// TIA Portal V19 export
FUNCTION_BLOCK "TYPIC_C103_IF_HVI"   // FB20, FBD
TITLE = TYPIC_C103_IF_HVI: ALSB
{ S7_Optimized_Access := 'TRUE' }
AUTHOR : OCOTECH
FAMILY : Typical
NAME : C103.701
// Logisch Object Besturing: C103.802
// 
// De interne functie laagspanningsverdeelbord verzorgt de bewaking van een laagspanningsverdeelbord.
// stored: MemoryReserve 10, SetENOAutomatically false
   VAR_INPUT
      EXT_AUT { ExternalAccessible := 'False'; ExternalVisible := 'False'; ExternalWritable := 'False'} : Bool;   // Externe (hoofd) beveiliging (1 = OK)
      EXT_HW { ExternalAccessible := 'False'; ExternalVisible := 'False'; ExternalWritable := 'False'} : Bool;   // Sturings hardware (PLC) bewaking (1 = OK)
      IN_PWR1 { ExternalAccessible := 'False'; ExternalVisible := 'False'; ExternalWritable := 'False'} : Real;   // Actief vermogen
      IN_PWR2 { ExternalAccessible := 'False'; ExternalVisible := 'False'; ExternalWritable := 'False'} : Real;   // Reactief vermogen
      IN_SPA_1 { ExternalAccessible := 'False'; ExternalVisible := 'False'; ExternalWritable := 'False'} : Real;   // Spanningsniveau lijn 1
      IN_SPA_2 { ExternalAccessible := 'False'; ExternalVisible := 'False'; ExternalWritable := 'False'} : Real;   // Spanningsniveau lijn 2
      IN_SPA_3 { ExternalAccessible := 'False'; ExternalVisible := 'False'; ExternalWritable := 'False'} : Real;   // Spanningsniveau lijn 3
      IN_SPA_4 { ExternalAccessible := 'False'; ExternalVisible := 'False'; ExternalWritable := 'False'} : Real;   // Lijnspanning L1-L2
      IN_SPA_5 { ExternalAccessible := 'False'; ExternalVisible := 'False'; ExternalWritable := 'False'} : Real;   // Lijnspanning L2-L3
      IN_SPA_6 { ExternalAccessible := 'False'; ExternalVisible := 'False'; ExternalWritable := 'False'} : Real;   // Lijnspanning L1-L3
      IN_STR_1 { ExternalAccessible := 'False'; ExternalVisible := 'False'; ExternalWritable := 'False'} : Real;   // Stroom lijn 1
      IN_STR_2 { ExternalAccessible := 'False'; ExternalVisible := 'False'; ExternalWritable := 'False'} : Real;   // Stroom lijn 2
      IN_STR_3 { ExternalAccessible := 'False'; ExternalVisible := 'False'; ExternalWritable := 'False'} : Real;   // Stroom lijn 3
      IN_STR_4 { ExternalAccessible := 'False'; ExternalVisible := 'False'; ExternalWritable := 'False'} : Real;   // Stroom nulleider
      IN_PHI { ExternalAccessible := 'False'; ExternalVisible := 'False'; ExternalWritable := 'False'} : Real;   // Arbeidsfactor
      IN_BEV_SPA { ExternalAccessible := 'False'; ExternalVisible := 'False'; ExternalWritable := 'False'} : Bool;   // Status beveiliging detectie railspanning
      IN_SPA2 { ExternalAccessible := 'False'; ExternalVisible := 'False'; ExternalWritable := 'False'} : Bool;   // Status detectie railspanning
      IN_SPA1_STO { ExternalAccessible := 'False'; ExternalVisible := 'False'; ExternalWritable := 'False'} : Bool;   // Status detectie railspanning
      IN_PHI_OK { ExternalAccessible := 'False'; ExternalVisible := 'False'; ExternalWritable := 'False'} : Bool;   // Status fasebewaking
      IN_HLP_OK { ExternalAccessible := 'False'; ExternalVisible := 'False'; ExternalWritable := 'False'} : Bool;   // Status hulpvoedingen (groepscontact)
      IN_SPD_OK { ExternalAccessible := 'False'; ExternalVisible := 'False'; ExternalWritable := 'False'} : Bool;   // Status overspanningsbeveiliging
      IN_SPA3_STO { ExternalAccessible := 'False'; ExternalVisible := 'False'; ExternalWritable := 'False'} : Bool;   // Status storing detectie railspanning
      IN_SPA4_STO { ExternalAccessible := 'False'; ExternalVisible := 'False'; ExternalWritable := 'False'} : Bool;   // Status storing detectie railspanning
      IN_STS1 { ExternalAccessible := 'False'; ExternalVisible := 'False'; ExternalWritable := 'False'} : Bool;   // Status van elke schuif [IN]
      IN_STS2 { ExternalAccessible := 'False'; ExternalVisible := 'False'; ExternalWritable := 'False'} : Bool;   // Status van elke schuif [TEST]
      IN_STS3 { ExternalAccessible := 'False'; ExternalVisible := 'False'; ExternalWritable := 'False'} : Bool;   // Status van elke schuif [UIT]
      IN_AUT_TOE { ExternalAccessible := 'False'; ExternalVisible := 'False'; ExternalWritable := 'False'} : Bool;   // Standmelding van elke vermogenschakelaar TOE [gesloten]
      IN_OK { ExternalAccessible := 'False'; ExternalVisible := 'False'; ExternalWritable := 'False'} : Bool;   // Standmelding beveiliging vertrek
   END_VAR
   VAR_OUTPUT
      VAR_IF_HVI { ExternalAccessible := 'False'; ExternalVisible := 'False'; ExternalWritable := 'False'} : "C103_VAR_IF_HVI_TYPIC";   // Struct met alle variabelen naar bovenliggende functies
   END_VAR
   VAR
      STO { ExternalWritable := 'False'} : Struct   // Storingen
         A001 { ExternalAccessible := 'False'; ExternalVisible := 'False'} : Bool;   // Laagspanningsverdeelbord beveiliging aangesproken
         A002 { ExternalAccessible := 'False'; ExternalVisible := 'False'} : Bool;   // Laagspanningsverdeelbord in storing
      END_STRUCT;
      VAR { ExternalWritable := 'False'} : Struct   // Variabelen
         PWR1 { ExternalAccessible := 'False'; ExternalVisible := 'False'} : Real;   // Actief vermogen
         PWR2 { ExternalAccessible := 'False'; ExternalVisible := 'False'} : Real;   // Reactief vermogen
         SPA_1 { ExternalAccessible := 'False'; ExternalVisible := 'False'} : Real;   // Spanningsniveau lijn 1
         SPA_2 { ExternalAccessible := 'False'; ExternalVisible := 'False'} : Real;   // Spanningsniveau lijn 2
         SPA_3 { ExternalAccessible := 'False'; ExternalVisible := 'False'} : Real;   // Spanningsniveau lijn 3
         SPA_4 { ExternalAccessible := 'False'; ExternalVisible := 'False'} : Real;   // Lijnspanning L1-L2
         SPA_5 { ExternalAccessible := 'False'; ExternalVisible := 'False'} : Real;   // Lijnspanning L2-L3
         SPA_6 { ExternalAccessible := 'False'; ExternalVisible := 'False'} : Real;   // Lijnspanning L1-L3
         STR_1 { ExternalAccessible := 'False'; ExternalVisible := 'False'} : Real;   // Stroom lijn 1
         STR_2 { ExternalAccessible := 'False'; ExternalVisible := 'False'} : Real;   // Stroom lijn 2
         STR_3 { ExternalAccessible := 'False'; ExternalVisible := 'False'} : Real;   // Stroom lijn 3
         STR_4 { ExternalAccessible := 'False'; ExternalVisible := 'False'} : Real;   // Stroom nulleider
         PHI { ExternalAccessible := 'False'; ExternalVisible := 'False'} : Real;   // Arbeidsfactor
         BEV_SPA { ExternalAccessible := 'False'; ExternalVisible := 'False'} : Bool;   // Status beveiliging detectie railspanning
         SPA2 { ExternalAccessible := 'False'; ExternalVisible := 'False'} : Bool;   // Status detectie railspanning
         SPA1_STO { ExternalAccessible := 'False'; ExternalVisible := 'False'} : Bool;   // Status detectie railspanning
         PHI_OK { ExternalAccessible := 'False'; ExternalVisible := 'False'} : Bool;   // Status fasebewaking
         HLP_OK { ExternalAccessible := 'False'; ExternalVisible := 'False'} : Bool;   // Status hulpvoedingen (groepscontact)
         SPD_OK { ExternalAccessible := 'False'; ExternalVisible := 'False'} : Bool;   // Status overspanningsbeveiliging
         SPA3_STO { ExternalAccessible := 'False'; ExternalVisible := 'False'} : Bool;   // Status storing detectie railspanning
         SPA4_STO { ExternalAccessible := 'False'; ExternalVisible := 'False'} : Bool;   // Status storing detectie railspanning
         STS1 { ExternalAccessible := 'False'; ExternalVisible := 'False'} : Bool;   // Status van elke schuif [IN]
         STS2 { ExternalAccessible := 'False'; ExternalVisible := 'False'} : Bool;   // Status van elke schuif [TEST]
         STS3 { ExternalAccessible := 'False'; ExternalVisible := 'False'} : Bool;   // Status van elke schuif [UIT]
         AUT_TOE { ExternalAccessible := 'False'; ExternalVisible := 'False'} : Bool;   // Standmelding van elke vermogenschakelaar TOE [gesloten]
         BEV_OK : Bool;
      END_STRUCT;
   END_VAR
BEGIN

REGION Network 1: START
END_REGION

REGION Network 2: +++ Verwerking meetwaarden en statussen +++
   // De meetwaarde en status wordt ontvangen vanuit de interne sturing.
END_REGION

REGION Network 3: +++ Storingen +++
   // Combinatie van de storingen
END_REGION

REGION Network 4: Storing A001: Laagspanningsverdeelbord beveiliging aangesproken
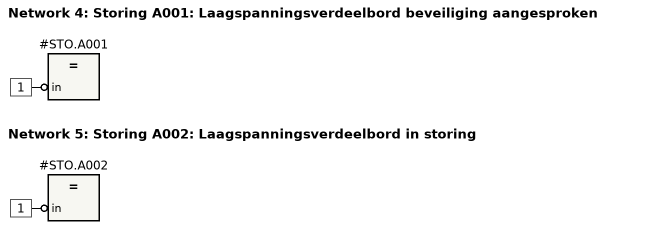
   #STO.A001 := NOT 1;
END_REGION

REGION Network 5: Storing A002: Laagspanningsverdeelbord in storing
   #STO.A002 := NOT 1;
END_REGION

REGION Network 6 (SCL): EINDE
   // Variabelen van intern scada rakvlak naar outputs copieren
   #VAR_IF_HVI.PWR1 := #VAR.PWR1;
   #VAR_IF_HVI.PWR2 := #VAR.PWR2;
   #VAR_IF_HVI.SPA_1 := #VAR.SPA_1;
   #VAR_IF_HVI.SPA_2 := #VAR.SPA_2;
   #VAR_IF_HVI.SPA_3 := #VAR.SPA_3;
   #VAR_IF_HVI.SPA_4 := #VAR.SPA_4;
   #VAR_IF_HVI.SPA_5 := #VAR.SPA_5;
   #VAR_IF_HVI.SPA_6 := #VAR.SPA_6;
   #VAR_IF_HVI.STR_1 := #VAR.STR_1;
   #VAR_IF_HVI.STR_2 := #VAR.STR_2;
   #VAR_IF_HVI.STR_3 := #VAR.STR_3;
   #VAR_IF_HVI.STR_4 := #VAR.STR_4;
   #VAR_IF_HVI.PHI := #VAR.PHI;
   #VAR_IF_HVI.BEV_SPA := #VAR.BEV_SPA;
   #VAR_IF_HVI.SPA2 := #VAR.SPA2;
   #VAR_IF_HVI.SPA1_STO := #VAR.SPA1_STO;
   #VAR_IF_HVI.PHI_OK := #VAR.PHI_OK;
   #VAR_IF_HVI.HLP_OK := #VAR.HLP_OK;
   #VAR_IF_HVI.SPD_OK := #VAR.SPD_OK;
   #VAR_IF_HVI.SPA3_STO := #VAR.SPA3_STO;
   #VAR_IF_HVI.SPA4_STO := #VAR.SPA4_STO;
   #VAR_IF_HVI.STS1 := #VAR.STS1;
   #VAR_IF_HVI.STS2 := #VAR.STS2;
   #VAR_IF_HVI.STS3 := #VAR.STS3;
   #VAR_IF_HVI.AUT_TOE := #VAR.AUT_TOE;
   #VAR_IF_HVI.BEV_OK := #VAR.BEV_OK;
END_REGION
END_FUNCTION_BLOCK
